{attribute 'qualified_only'}
{attribute 'strict'}
TYPE E_UserGroup :
(
	Admin := 0,
    Operator := 1,
    Guest := 2
);
END_TYPE

(* stored: Version 1.1.0.1, ProductVersion 3.1.4024.12
   DUT E_UserGroup: Id {ee6a2da3-1b1b-42f5-aa70-b7649e6f1667} *)
